FUNCTION_BLOCK PUBLIC FB_Decorator IMPLEMENTS I_Pizza
VAR_INPUT
END_VAR
VAR_OUTPUT
END_VAR
VAR
	ipSideOrder	: I_Pizza;
END_VAR

METHOD FB_init : BOOL
VAR_INPUT
	bInitRetains	: BOOL; // if TRUE, the retain variables are initialized (warm start / cold start)
	bInCopyCode		: BOOL;  // if TRUE, the instance afterwards gets moved into the copy code (online change)
	ipSideOrder		: I_Pizza;
END_VAR
THIS^.ipSideOrder := ipSideOrder;
END_METHOD

{warning 'add method implementation'}
METHOD GetDescription : STRING
END_METHOD

{warning 'add method implementation'}
METHOD GetPrice : LREAL
END_METHOD

PROPERTY PUBLIC ipDecorator : I_Pizza
GET
ipDecorator := THIS^.ipSideOrder;
END_GET
SET
THIS^.ipSideOrder := ipDecorator;
END_SET
END_PROPERTY

END_FUNCTION_BLOCK

(* stored: Version 1.1.0.1, ProductVersion 3.1.4022.16
   POU FB_Decorator: Id {bfa4a11a-0c97-446f-a048-14209d21dc7f}, SpecialFunc None
   Method FB_init: Id {f860e243-06dc-4c02-b222-b90e3c814283}
   Method GetDescription: Id {f850d087-7b0d-4744-98fa-824641fa0d67}
   Method GetPrice: Id {08a19f83-703c-4c0a-80fe-893334fb7c30}
   Property ipDecorator: Id {c618fb2b-b304-47b4-b86e-e54401a158b5}
   Get Get: Id {2c71dc2a-41ac-4e73-bdb1-25079fa15bcc}
   Set Set: Id {d1ef92e7-23d1-4085-8594-79a261019e21} *)
